FUNCTION_BLOCK Model
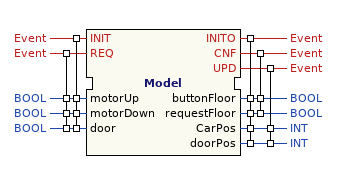
  EVENT_INPUT
    INIT WITH motorUp, motorDown, door;
    REQ WITH motorUp, motorDown, door;
  END_EVENT
  EVENT_OUTPUT
    INITO WITH buttonFloor, requestFloor, CarPos, doorPos;
    CNF WITH buttonFloor, requestFloor;
    UPD WITH CarPos, doorPos;
  END_EVENT
  VAR_INPUT
    motorUp : BOOL;
    motorDown : BOOL;
    door : BOOL;
  END_VAR
  VAR_OUTPUT
    buttonFloor : BOOL;
    requestFloor : BOOL;
    CarPos : INT;
    doorPos : INT;
  END_VAR
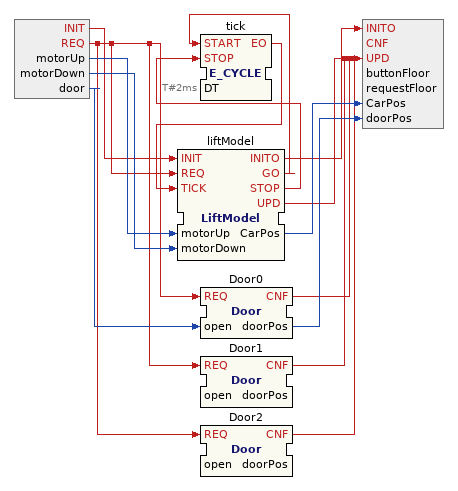
  FBS
    tick : E_CYCLE(DT := T#2ms);
    liftModel : LiftModel;
    Door0 : Door;
    Door1 : Door;
    Door2 : Door;
  END_FBS
  EVENT_CONNECTIONS
    INIT TO liftModel.INIT;
    REQ TO liftModel.REQ;
    tick.EO TO liftModel.TICK;
    liftModel.GO TO tick.START;
    liftModel.STOP TO tick.STOP;
    liftModel.UPD TO UPD;
    liftModel.INITO TO INITO;
    Door0.CNF TO UPD;
    REQ TO Door0.REQ;
    Door1.CNF TO UPD;
    Door2.CNF TO UPD;
    REQ TO Door1.REQ;
    REQ TO Door2.REQ;
  END_CONNECTIONS
  DATA_CONNECTIONS
    motorUp TO liftModel.motorUp;
    motorDown TO liftModel.motorDown;
    liftModel.CarPos TO CarPos;
    Door0.doorPos TO doorPos;
    door TO Door0.open;
  END_CONNECTIONS
END_FUNCTION_BLOCK
